// TIA Portal V16 export
// export: Created 2021-07-12T14:47:21.3062335Z, ExportSetting WithDefaults, DisplayName Totally Integrated Automation Portal, DisplayVersion V16, DisplayName TIA Portal Version Control Interface, DisplayVersion V16, DisplayName TIA Portal Openness, DisplayVersion V16, DisplayName STEP 7 Professional, DisplayVersion V16, DisplayName STEP 7 Safety, DisplayVersion V16, DisplayName WinCC Professional, DisplayVersion V16
TYPE "SimaHydTO_typeHMIConnectionParameterSettingsStatus"
TITLE = SimaHydTO_typeHMIConnectionParameterSettingsStatus
// HMI interface: Parameter settings - Status (PLC -> HMI)
// stored: IsFailsafeCompliant false
   STRUCT
      EditorActive : Bool;
      StateActivation : Int;   // 0: none / 1: activated / 2: error
      StateSaving : Int;   // 0: none / 1: saved / 2: error
      StateLoading : Int;   // 0: none / 1: restoreded / 2: error
      VCharSelector { S7_SetPoint := 'True'} : "SimaHydTO_typeHMIConnectionVCharSelectorStatus";
   END_STRUCT;
END_TYPE
